TEXTLIST TextList_UVLed_state
  0 = 'off'
  1 = 'initializing'
  2 = 'ready'
  3 = 'applying_settings'
  4 = 'settings_applied'
  10 = 'ready_for_curing'
  5 = 'curing'
  6 = 'setting_off'
  100 = 'error'
   = ''
END_TEXTLIST

(* stored: Version 1.1.0.1, ProductVersion 3.1.4024.11
   TextList TextList_UVLed_state: Id {9c1df7cd-034e-413b-b150-8ff2d036fe54} *)
